// TwinCAT 3 PLC project MQTT
// ProgramVersion: 3.1.4024.0
// libraries:
//   Tc2_BA, * (Beckhoff Automation GmbH)
//   Tc2_BABasic, * (Beckhoff Automation GmbH)
//   Tc2_DALI, * (Beckhoff Automation GmbH)
//   Tc2_Standard, * (Beckhoff Automation GmbH)
//   Tc2_System, * (Beckhoff Automation GmbH)
//   Tc2_Utilities, * (Beckhoff Automation GmbH)
//   Tc3_IotBase, * (Beckhoff Automation GmbH)
//   Tc3_JsonXml, * (Beckhoff Automation GmbH)
//   Tc3_Module, * (Beckhoff Automation GmbH)
// project tree:
//   / PlcTask.TcTTO
//   POUs/Bediening/ FB_Drukknoppen.TcPOU, FB_Sensor.TcPOU, FB_Verbruikmeter.TcPOU, Verbruik_input.TcDUT
//   POUs/ FB_Licht_withFeedback.TcPOU, FB_Light.TcPOU (excluded from build), AchtB.TcPOU, PrgMqttCom.TcPOU
//   POUs/Gebruiker/ FB_Dakraam.TcPOU, FB_Garagepoort.TcPOU, FB_Stopcontact.TcPOU, FB_Warmtepomp.TcPOU, Licht_output.TcDUT, Stopcontact_output.TcDUT, Warmtepomp_Signalen.TcDUT
//   POUs/Kamers/ FB_Eethoek.TcPOU, FB_Slaapkamer.TcPOU, FB_Tuin.TcPOU, FB_Zithoek.TcPOU
//   POUs/Verdieping/ FB_Garage.TcPOU, FB_Gelijkvloers.TcPOU, FB_Slaapkamers.TcPOU, FB_Technische_ruimte.TcPOU
// real-time tasks:
//   TASK PlcTask: cycle T#10ms, priority 20, ADS port 350

CONFIGURATION MQTT
    RESOURCE PLC ON TwinCAT3
        TASK PlcTask(INTERVAL := T#10ms, PRIORITY := 20);
        PROGRAM AchtB WITH PlcTask : AchtB;
    END_RESOURCE
END_CONFIGURATION

// ---- POUs/Bediening/Verbruik_input.TcDUT
TYPE Verbruik_input :
STRUCT
	Puls		AT %I*	: BOOL;
	Value				: REAL;
//	Meetgegevens		: ST_Meetgegevens;
END_STRUCT
END_TYPE

// ---- POUs/Gebruiker/Licht_output.TcDUT
TYPE Licht_output :
STRUCT
	bOutput		AT %Q*	: BOOL;
	nLicht		AT %Q*	: INT;
	feedback_licht		: INT;
	status_licht		: BOOL;
	Inschakeltijd		: REAL;
	
END_STRUCT
END_TYPE

// ---- POUs/Gebruiker/Stopcontact_output.TcDUT
TYPE Stopcontact_output  EXTENDS Licht_output :
STRUCT
	Verbruik	: REAL;
	Vermogen	: REAL;
	
END_STRUCT
END_TYPE

// ---- POUs/Gebruiker/Warmtepomp_Signalen.TcDUT
TYPE Warmtepomp_Signalen :
STRUCT
	laagtarief			AT %Q*	: BOOL;
	piekvermogen_uit	AT %Q*	: BOOL;
END_STRUCT
END_TYPE

// ---- POUs/AchtB.TcPOU
PROGRAM AchtB
VAR
	Woonruimte			: FB_Gelijkvloers;
	Tuin				: FB_Tuin;
	Slaapkamers			: FB_Slaapkamers;
	Garage				: FB_Garage;
	Technische_ruimte	: FB_Technische_ruimte;
	
END_VAR

PrgMqttCom();

END_PROGRAM

// ---- POUs/Verdieping/FB_Gelijkvloers.TcPOU
FUNCTION_BLOCK FB_Gelijkvloers
VAR
	Bediening_Keuken	: FB_Drukknoppen;
	Bediening_Inkom		: FB_Drukknoppen;
	Bediening_eethoek	: FB_Drukknoppen;
	Bediening_zithoek	: FB_Drukknoppen;
	
	Beweging_Wasplaats	: FB_Sensor;
	Beweging_WC			: FB_Sensor;
	Beweging_Keuken		: FB_Sensor;
	
	Keuken				: FB_StairwellLight;
	Wasplaats			: FB_StairwellLight;
	WC_onder			: FB_StairwellLight;
	Eethoek				: FB_Eethoek;
	Zithoek				: FB_Zithoek;
	Vide				: FB_Dimmer1Switch;
	
	licht_keuken		: Licht_output;
	licht_wasplaats		: Licht_output;
	licht_wc_onder		: Licht_output;
	licht_vide			: Licht_output;

END_VAR

END_FUNCTION_BLOCK

// ---- POUs/Bediening/FB_Drukknoppen.TcPOU
FUNCTION_BLOCK FB_Drukknoppen
VAR
	Input		AT %I*	: ARRAY [1..6] OF BOOL;
	Short_Long			: ARRAY [1..6] OF FB_ShortLongClick;
	Single_Double		: ARRAY [1..6] OF FB_SingleDoubleClick;

END_VAR

END_FUNCTION_BLOCK

// ---- POUs/Bediening/FB_Sensor.TcPOU
FUNCTION_BLOCK FB_Sensor
VAR
	bInput		AT %I*	: BOOL;
	nInput		AT %I*	: BOOL;
	
END_VAR

END_FUNCTION_BLOCK

// ---- POUs/Kamers/FB_Eethoek.TcPOU
FUNCTION_BLOCK FB_Eethoek
VAR
	bediening_eethoek	: FB_Drukknoppen;
	
	Eettafel			: FB_Dimmer1Switch;
	Foto_papa			: FB_DALIV2Dimmer1Switch;
	Foto_whiskey		: FB_DALIV2Dimmer1Switch;
	Brutale_L			: FB_DALIV2Dimmer1Switch;
	Brutale_R			: FB_DALIV2Dimmer1Switch;
	Scene_Eethoek		: FB_ScenesLighting;

	licht_tafel			: Licht_output;
	licht_Foto_papa		: Licht_output;
	licht_Foto_whiskey  : Licht_output;
    licht_Brutale_L	    : Licht_output;
    licht_Brutale_R	    : Licht_output;
	
END_VAR

END_FUNCTION_BLOCK

// ---- POUs/Kamers/FB_Zithoek.TcPOU
FUNCTION_BLOCK FB_Zithoek
VAR
	Zithoek_LV			: FB_DALIV2Dimmer1Switch;
	Zithoek_RV			: FB_DALIV2Dimmer1Switch;
	Zithoek_LA			: FB_DALIV2Dimmer1Switch;
	Zithoek_MA			: FB_DALIV2Dimmer1Switch;
	Zithoek_RA			: FB_DALIV2Dimmer1Switch;

	licht_Zithoek_LV	: Licht_output;
	licht_Zithoek_RV	: Licht_output;
	licht_Zithoek_LA	: Licht_output;
	licht_Zithoek_MA	: Licht_output;
	licht_Zithoek_RA	: Licht_output;

END_VAR

END_FUNCTION_BLOCK

// ---- POUs/Kamers/FB_Tuin.TcPOU
FUNCTION_BLOCK FB_Tuin
VAR
	Beweging_inrit	: FB_Sensor;
	
	vijver			: FB_Light;
	tuin			: FB_Light;
	hondenhok		: FB_Light;
	weide			: FB_Light;
	inrit			: FB_Light;
	terras			: FB_Dimmer1Switch;
	barruimte		: ARRAY [1..4] OF FB_DALIV2Dimmer1Switch;
	brievenbus		: ARRAY [1..4] OF FB_DALIV2Dimmer1Switch;
	
	licht_vijver	: Licht_output;
	licht_tuin		: Licht_output;
	licht_hondenhok	: Licht_output;
	licht_weide		: Licht_output;
	licht_inrit		: Licht_output;
	licht_terras	: Licht_output;
	licht_barruimte	: Licht_output;
	licht_brievenbus: Licht_output;
	
	stopcontact_vijverpomp	: FB_Stopcontact;
	stopcontact_UV_lamp		: FB_Stopcontact;
	stopcontact_vijverlucht	: FB_Stopcontact;
	stopcontacten_tuin		: FB_Stopcontact;
	
END_VAR

END_FUNCTION_BLOCK

// ---- POUs/FB_Light.TcPOU
FUNCTION_BLOCK FB_Light
VAR
	licht		AT %Q*	: BOOL;
END_VAR

METHOD Turn_off : BOOL
VAR_INPUT
END_VAR
licht	:= FALSE;
END_METHOD

METHOD Turn_on : BOOL
VAR_INPUT
END_VAR
licht	:= TRUE;
END_METHOD

END_FUNCTION_BLOCK

// ---- POUs/Gebruiker/FB_Stopcontact.TcPOU
FUNCTION_BLOCK FB_Stopcontact
VAR
	Output			: Stopcontact_output;
	kWh_meter		: FB_Verbruikmeter;
	
END_VAR

END_FUNCTION_BLOCK

// ---- POUs/Bediening/FB_Verbruikmeter.TcPOU
FUNCTION_BLOCK FB_Verbruikmeter
VAR
	Meetsignaal	: Verbruik_input;
	
END_VAR

END_FUNCTION_BLOCK

// ---- POUs/Verdieping/FB_Slaapkamers.TcPOU
FUNCTION_BLOCK FB_Slaapkamers
VAR
	bediening_badkmaer	: FB_Drukknoppen;
	sensor_nachthal		: FB_sensor;
	sensor_traphal		: FB_Sensor;
	
	master_slaapkamer	: FB_Slaapkamer;
	linnea_slaapkamer	: FB_Slaapkamer;
	dakraam_links		: FB_Dakraam;
	dakraam_rechts		: FB_Dakraam;

	Nachthal			: FB_StairwellDimmer;
	Traphal				: FB_StairwellDimmer;
	Badkamer			: FB_Light;
	Badkamer_spiegel	: FB_Light;

	licht_nachthal		: Licht_output;
	licht_traphal		: Licht_output;
	licht_badkamer		: Licht_output;
	licht_spiegel		: Licht_output;
	
END_VAR

END_FUNCTION_BLOCK

// ---- POUs/Kamers/FB_Slaapkamer.TcPOU
FUNCTION_BLOCK FB_Slaapkamer
VAR
	bediening_bed_L		: FB_Drukknoppen;
	bediening_bed_R		: FB_Drukknoppen;
	bediening_deur		: FB_Drukknoppen;
	
	Verlichting			: FB_Dimmer1Switch;
	Verlichting_bureau	: FB_Dimmer1Switch;
	Verlichting_bed		: FB_Dimmer1Switch;
	
	licht				: Licht_output;
	licht_bureau		: Licht_output;
	licht_bed			: Licht_output;
	
END_VAR

END_FUNCTION_BLOCK

// ---- POUs/Gebruiker/FB_Dakraam.TcPOU
FUNCTION_BLOCK FB_Dakraam
VAR_INPUT
END_VAR
VAR_OUTPUT
END_VAR
VAR
END_VAR

END_FUNCTION_BLOCK

// ---- POUs/Verdieping/FB_Garage.TcPOU
FUNCTION_BLOCK FB_Garage
VAR
	Bediening_deur			: FB_Drukknoppen;
	Bediening_werkruimte	: FB_Drukknoppen;
	Garage_links			: FB_StairwellLight;
	Garage_rechts			: FB_StairwellLight;
	Garagepoort				: ARRAY [1..4] OF FB_DALIV2Dimmer1Switch;
	Leeuw					: ARRAY [1..4] OF FB_DALIV2Dimmer1Switch;
	
	Poortopener				: FB_Garagepoort;
	Elektriciteitsmeter		: FB_Verbruikmeter;
	Leidingwater			: FB_Verbruikmeter;
	Regenwater				: FB_Verbruikmeter;
//	Regenwaterput			: FB_niveaumeter;
	
	licht_Garage_l			: Licht_output;
	licht_Garage_r			: Licht_output;
	licht_Garagepoort		: Licht_output;
	licht_Leeuw				: Licht_output;
	
END_VAR

END_FUNCTION_BLOCK

// ---- POUs/Gebruiker/FB_Garagepoort.TcPOU
FUNCTION_BLOCK FB_Garagepoort
VAR_INPUT
END_VAR
VAR_OUTPUT
END_VAR
VAR
END_VAR

END_FUNCTION_BLOCK

// ---- POUs/Verdieping/FB_Technische_ruimte.TcPOU
FUNCTION_BLOCK FB_Technische_ruimte
VAR
	Bediening_TR	: FB_Drukknoppen;
	
	TR_verlichting	: FB_StairwellLight;
	
	licht_TR		: licht_output;
	
	zonnepanelen	: FB_Verbruikmeter;
	warmtepomp		: FB_Warmtepomp;
// 	ventilatie

END_VAR

END_FUNCTION_BLOCK

// ---- POUs/Gebruiker/FB_Warmtepomp.TcPOU
FUNCTION_BLOCK FB_Warmtepomp
VAR
	Verbruik		: FB_Verbruikmeter;
	Communicatie	: Warmtepomp_Signalen;
	
END_VAR

END_FUNCTION_BLOCK

// ---- POUs/PrgMqttCom.TcPOU
PROGRAM PrgMqttCom
VAR
	fbMqttClient : FB_IotMqttClient;
	bSetParameter : BOOL := TRUE;
	bConnect 	: BOOL := TRUE;
	Host_ip		: STRING(13) := '192.168.0.190';
	Host_port	: UINT  := 1883;
	(* published message *)
	sTopicPub : STRING(255) := 'homeassistant';
	sPayloadPub : STRING(255);
	i: UDINT;
	fbTimer : TON := (PT:=T#1S);
	
	(* received message *)
	bSubscribed : BOOL;
	sTopicSub : STRING(255) := 'homeassistant';
	{attribute 'TcEncoding':='UTF-8'}
	sTopicRcv : STRING(255);
	{attribute 'TcEncoding':='UTF-8'}
	sPayloadRcv : STRING(255);
	fbMessageQueue : FB_IotMqttMessageQueue;
	fbMessage : FB_IotMqttMessage;
	
	hrErrorOccurred : HRESULT; // contains the latest occurred error
	timer	: BOOL;
END_VAR

IF bSetParameter THEN
	bSetParameter := FALSE;
	fbMqttClient.sHostName:= Host_ip;
	fbMqttClient.nHostPort:= Host_port;
//	fbMqttClient.sClientId:= 'MyTcMqttClient'; 
	fbMqttClient.sTopicPrefix:= ''; 
//	fbMqttClient.nKeepAlive:= 60; 
//	fbMqttClient.sUserName:= ;
//	fbMqttClient.sUserPassword:= ; 
//	fbMqttClient.stWill:= ; 
//	fbMqttClient.stTLS:= ;
	fbMqttClient.ipMessageQueue := fbMessageQueue;
END_IF

fbMqttClient.Execute(bConnect);
IF fbMqttClient.bError THEN
	// add your error logging here
	hrErrorOccurred := fbMqttClient.hrErrorCode;
END_IF

IF fbMessageQueue.nQueuedMessages > 0 THEN
	IF fbMessageQueue.Dequeue(fbMessage:=fbMessage) THEN
		fbMessage.GetTopic(pTopic:=ADR(sTopicRcv), nTopicSize:=SIZEOF(sTopicRcv) );
		fbMessage.GetPayload(pPayload:=ADR(sPayloadRcv), nPayloadSize:=SIZEOF(sPayloadRcv), bSetNullTermination := TRUE);
	END_IF
END_IF

IF fbMqttClient.bConnected THEN
	IF NOT bSubscribed THEN
		bSubscribed := fbMqttClient.Subscribe(sTopic:=sTopicSub, eQoS:=TcIotMqttQos.AtLeastOnceDelivery);
		IF fbMqttClient.bError THEN
			// add your error logging here
			hrErrorOccurred := fbMqttClient.hrErrorCode;
		END_IF
	END_IF
	fbTimer(IN:=timer);
	IF fbTimer.Q THEN // publish new payload every second
		fbTimer(IN:=FALSE);
		i := i + 1;
		sPayloadPub := CONCAT('MyMessage', TO_STRING(i));
		fbMqttClient.Publish(	sTopic:= sTopicPub, 
								pPayload:= ADR(sPayloadPub), nPayloadSize:= LEN2(ADR(sPayloadPub))+1, 
								eQoS:= TcIotMqttQos.AtLeastOnceDelivery, bRetain:= TRUE, bQueue:= FALSE );
		IF fbMqttClient.bError THEN
			// add your error logging here
			hrErrorOccurred := fbMqttClient.hrErrorCode;
		END_IF
	END_IF
END_IF

END_PROGRAM

// ---- POUs/FB_Licht_withFeedback.TcPOU
FUNCTION_BLOCK FB_Licht_withFeedback EXTENDS FB_Light
VAR
END_VAR

PROPERTY Light_is_off : bool
GET
IF NOT SUPER^.licht THEN
	Light_is_off	:= TRUE;
	
ELSE
	Light_is_off	:= FALSE;
	
END_IF
END_GET
END_PROPERTY

PROPERTY Light_is_on : bool
GET
IF SUPER^.licht THEN
	Light_is_on	:= TRUE;
	
ELSE
	Light_is_on	:= FALSE;
	
END_IF
END_GET
END_PROPERTY

END_FUNCTION_BLOCK
